Staubli VAL3: stop.pgx

program stop()
begin
  bRunning = false
  taskKill("mainLoop")
end
